// TwinCAT 3 PLC project PLC_SerialCom_Sample1
// ProgramVersion: 3.1.0.8
// libraries:
//   Tc2_SerialCom, * (Beckhoff Automation GmbH)
//   Tc2_Standard, * (Beckhoff Automation GmbH)
//   Tc3_Module, * (Beckhoff Automation GmbH)
// project tree:
//   GVLs/ gc.TcGVL, GVL.TcGVL
//   / PlcTask_Fast.TcTTO (not stored), PlcTask_Standard.TcTTO
//   POUs/ Background.TcPOU, BackgroundKL.TcPOU, BackgroundEL.TcPOU, FB_SerialCom.TcPOU, MAIN.TcPOU, BackgroundPcCOM.TcPOU (not stored), test.TcPOU
// real-time tasks:
//   TASK PlcTask_Fast: cycle T#2ms, priority 19, ADS port 350
//   TASK PlcTask_Standard: cycle T#10ms, priority 20, ADS port 351
// motion (NC):
//   TASK NC-Task 1 SAF: cycle T#2ms, priority 4, ADS port 501
//   TASK NC-Task 1 SVB: cycle T#10ms, priority 8, ADS port 511
//   AXIS Axis 1 (id 1)
//     OtherSettings: AllowMotionCmdToSlave=true
//     encoder EncType=19
//       EncPara: MaxCount=#xffffffff
//     drive DrvType=16
//       DrvPara: MaxCount=#xffffffff, DriveControlDWord=#x00020000
//         Analog: TorqueSetpointScale=10, ScaleFactorActTorque=0.1
//         TimeComp: TaskDelayCycles=1
//     controller CtrType=1
//       CtrPara: PriorControlFactor=1
//         Observer: BandWidth=20
//   AXIS Axis 2 (id 2)
//     OtherSettings: AllowMotionCmdToSlave=true
//     encoder EncType=19
//       EncPara: MaxCount=#xffffffff
//     drive DrvType=16
//       DrvPara: MaxCount=#xffffffff, DriveControlDWord=#x00020000
//         Analog: TorqueSetpointScale=10, ScaleFactorActTorque=0.1
//         TimeComp: TaskDelayCycles=1
//     controller CtrType=1
//       CtrPara: PriorControlFactor=1
//         Observer: BandWidth=20
// I/O:
//   DEVICE Device 1 (COM Port) (disabled)
//   DEVICE Device 3 (EtherCAT) (disabled), AmsNetId 172.17.60.154.4.1
//     Term 1 (EK1100) [EK1100 EtherCAT Coupler (2A E-Bus)]
//       Term 2 (EL6001) [EL6001 Interface (RS232)]
//       Box 3 (BK1250)
//   DEVICE Device 2 (EtherCAT), AmsNetId 192.168.2.2.3.1
//     Term 4 (EK1914) [EK1914, 2 Ch. Safety Input/Output 24V,  TwinSAFE]
//       modules: Module 1 (FSOE), Module 2 (DIO)
//       Term 5 (EL9410) [EL9410 E-Bus Power Supplier  (Diagnostics)]
//       Term 6 (EL3164) [EL3164 4Ch. Ana. Input 0-10V]
//       Term 7 (EL4104) [EL4104 4Ch. Ana. Output 0-10V, 16bit]
//       Term 5 (EL6614) [EL6614 4 Port Switch (Ethernet, CoE)]
//       Term 9 (EL6002) [EL6002 Interface 2Ch. (RS232)]
//       Term 10 (EL9410) [EL9410 E-Bus Power Supplier  (Diagnostics)]
//       Term 11 (EL7201-9014) [EL7201-9014 1Ch. MDP742 Servo motor output stage with OCT (50V, 2.8A RMS) and STO input]
//       Term 12 (EL7201-9014) [EL7201-9014 1Ch. MDP742 Servo motor output stage with OCT (50V, 2.8A RMS) and STO input]
//       Term 10 (EL9011) [EL9011 End Terminal]
// variable links:
//   NC-Task 1 SAF/Axes/Axis 1 <-> Device 2 (EtherCAT)/Term 4 (EK1914)/Term 11 (EL7201-9014)
//     Drive/Inputs/In/nDcOutputTime <-> InfoData/DcOutputShift
//     Drive/Inputs/In/nState1 <-> DRV Statusword/Statusword
//     Drive/Inputs/In/nState2 <-> DRV Statusword/Statusword @bit 8
//     Drive/Inputs/In/nState4 @bit 1 <-> WcState/InputToggle
//     Drive/Inputs/In/nState4 <-> WcState/WcState
//     Drive/Outputs/Out/nCtrl1 <-> DRV Controlword/Controlword
//     Drive/Outputs/Out/nCtrl2 <-> DRV Controlword/Controlword @bit 8
//     Drive/Outputs/Out/nDataOut2 <-> DRV Target velocity/Target velocity
//     Enc/Inputs/In/nDataIn1 <-> FB Position/Position
//     Enc/Inputs/In/nDcInputTime <-> InfoData/DcInputShift
//     Enc/Inputs/In/nState4 @bit 1 <-> WcState/InputToggle
//     Enc/Inputs/In/nState4 <-> WcState/WcState
//   NC-Task 1 SAF/Axes/Axis 2 <-> Device 2 (EtherCAT)/Term 4 (EK1914)/Term 12 (EL7201-9014)
//     Drive/Inputs/In/nDcOutputTime <-> InfoData/DcOutputShift
//     Drive/Inputs/In/nState1 <-> DRV Statusword/Statusword
//     Drive/Inputs/In/nState2 <-> DRV Statusword/Statusword @bit 8
//     Drive/Inputs/In/nState4 @bit 1 <-> WcState/InputToggle
//     Drive/Inputs/In/nState4 <-> WcState/WcState
//     Drive/Outputs/Out/nCtrl1 <-> DRV Controlword/Controlword
//     Drive/Outputs/Out/nCtrl2 <-> DRV Controlword/Controlword @bit 8
//     Drive/Outputs/Out/nDataOut2 <-> DRV Target velocity/Target velocity
//     Enc/Inputs/In/nDataIn1 <-> FB Position/Position
//     Enc/Inputs/In/nDcInputTime <-> InfoData/DcInputShift
//     Enc/Inputs/In/nState4 @bit 1 <-> WcState/InputToggle
//     Enc/Inputs/In/nState4 <-> WcState/WcState
//   PLC_SerialCom_Sample1/PLC_SerialCom_Sample1 Instance <-> Device 2 (EtherCAT)/Term 4 (EK1914)
//     PlcTask_Standard Inputs/test.xTestInput <-> Module 2 (DIO)/DIO Inputs/Input 1
//   PLC_SerialCom_Sample1/PLC_SerialCom_Sample1 Instance <-> Device 2 (EtherCAT)/Term 4 (EK1914)/Term 9 (EL6002)
//     PlcTask_Fast Inputs/BackgroundEL.astIn_EL6002[0]/D <-> COM TxPDO-Map Inputs Channel 1/Data In 0
//     PlcTask_Fast Inputs/BackgroundEL.astIn_EL6002[1]/D <-> COM TxPDO-Map Inputs Channel 2/Data In 0
//     PlcTask_Fast Inputs/BackgroundEL.astIn_EL6002[0]/D @bit 8 <-> COM TxPDO-Map Inputs Channel 1/Data In 1
//     PlcTask_Fast Inputs/BackgroundEL.astIn_EL6002[0]/D @bit 80 <-> COM TxPDO-Map Inputs Channel 1/Data In 10
//     PlcTask_Fast Inputs/BackgroundEL.astIn_EL6002[0]/D @bit 88 <-> COM TxPDO-Map Inputs Channel 1/Data In 11
//     PlcTask_Fast Inputs/BackgroundEL.astIn_EL6002[0]/D @bit 96 <-> COM TxPDO-Map Inputs Channel 1/Data In 12
//     PlcTask_Fast Inputs/BackgroundEL.astIn_EL6002[0]/D @bit 104 <-> COM TxPDO-Map Inputs Channel 1/Data In 13
//     PlcTask_Fast Inputs/BackgroundEL.astIn_EL6002[0]/D @bit 112 <-> COM TxPDO-Map Inputs Channel 1/Data In 14
//     PlcTask_Fast Inputs/BackgroundEL.astIn_EL6002[0]/D @bit 120 <-> COM TxPDO-Map Inputs Channel 1/Data In 15
//     PlcTask_Fast Inputs/BackgroundEL.astIn_EL6002[0]/D @bit 128 <-> COM TxPDO-Map Inputs Channel 1/Data In 16
//     PlcTask_Fast Inputs/BackgroundEL.astIn_EL6002[0]/D @bit 136 <-> COM TxPDO-Map Inputs Channel 1/Data In 17
//     PlcTask_Fast Inputs/BackgroundEL.astIn_EL6002[0]/D @bit 144 <-> COM TxPDO-Map Inputs Channel 1/Data In 18
//     PlcTask_Fast Inputs/BackgroundEL.astIn_EL6002[0]/D @bit 152 <-> COM TxPDO-Map Inputs Channel 1/Data In 19
//     PlcTask_Fast Inputs/BackgroundEL.astIn_EL6002[0]/D @bit 16 <-> COM TxPDO-Map Inputs Channel 1/Data In 2
//     PlcTask_Fast Inputs/BackgroundEL.astIn_EL6002[0]/D @bit 160 <-> COM TxPDO-Map Inputs Channel 1/Data In 20
//     PlcTask_Fast Inputs/BackgroundEL.astIn_EL6002[0]/D @bit 168 <-> COM TxPDO-Map Inputs Channel 1/Data In 21
//     PlcTask_Fast Inputs/BackgroundEL.astIn_EL6002[0]/D @bit 24 <-> COM TxPDO-Map Inputs Channel 1/Data In 3
//     PlcTask_Fast Inputs/BackgroundEL.astIn_EL6002[0]/D @bit 32 <-> COM TxPDO-Map Inputs Channel 1/Data In 4
//     PlcTask_Fast Inputs/BackgroundEL.astIn_EL6002[0]/D @bit 40 <-> COM TxPDO-Map Inputs Channel 1/Data In 5
//     PlcTask_Fast Inputs/BackgroundEL.astIn_EL6002[0]/D @bit 48 <-> COM TxPDO-Map Inputs Channel 1/Data In 6
//     PlcTask_Fast Inputs/BackgroundEL.astIn_EL6002[0]/D @bit 56 <-> COM TxPDO-Map Inputs Channel 1/Data In 7
//     PlcTask_Fast Inputs/BackgroundEL.astIn_EL6002[0]/D @bit 64 <-> COM TxPDO-Map Inputs Channel 1/Data In 8
//     PlcTask_Fast Inputs/BackgroundEL.astIn_EL6002[0]/D @bit 72 <-> COM TxPDO-Map Inputs Channel 1/Data In 9
//     PlcTask_Fast Inputs/BackgroundEL.astIn_EL6002[1]/D @bit 8 <-> COM TxPDO-Map Inputs Channel 2/Data In 1
//     PlcTask_Fast Inputs/BackgroundEL.astIn_EL6002[1]/D @bit 80 <-> COM TxPDO-Map Inputs Channel 2/Data In 10
//     PlcTask_Fast Inputs/BackgroundEL.astIn_EL6002[1]/D @bit 88 <-> COM TxPDO-Map Inputs Channel 2/Data In 11
//     PlcTask_Fast Inputs/BackgroundEL.astIn_EL6002[1]/D @bit 96 <-> COM TxPDO-Map Inputs Channel 2/Data In 12
//     PlcTask_Fast Inputs/BackgroundEL.astIn_EL6002[1]/D @bit 104 <-> COM TxPDO-Map Inputs Channel 2/Data In 13
//     PlcTask_Fast Inputs/BackgroundEL.astIn_EL6002[1]/D @bit 112 <-> COM TxPDO-Map Inputs Channel 2/Data In 14
//     PlcTask_Fast Inputs/BackgroundEL.astIn_EL6002[1]/D @bit 120 <-> COM TxPDO-Map Inputs Channel 2/Data In 15
//     PlcTask_Fast Inputs/BackgroundEL.astIn_EL6002[1]/D @bit 128 <-> COM TxPDO-Map Inputs Channel 2/Data In 16
//     PlcTask_Fast Inputs/BackgroundEL.astIn_EL6002[1]/D @bit 136 <-> COM TxPDO-Map Inputs Channel 2/Data In 17
//     PlcTask_Fast Inputs/BackgroundEL.astIn_EL6002[1]/D @bit 144 <-> COM TxPDO-Map Inputs Channel 2/Data In 18
//     PlcTask_Fast Inputs/BackgroundEL.astIn_EL6002[1]/D @bit 152 <-> COM TxPDO-Map Inputs Channel 2/Data In 19
//     PlcTask_Fast Inputs/BackgroundEL.astIn_EL6002[1]/D @bit 16 <-> COM TxPDO-Map Inputs Channel 2/Data In 2
//     PlcTask_Fast Inputs/BackgroundEL.astIn_EL6002[1]/D @bit 160 <-> COM TxPDO-Map Inputs Channel 2/Data In 20
//     PlcTask_Fast Inputs/BackgroundEL.astIn_EL6002[1]/D @bit 168 <-> COM TxPDO-Map Inputs Channel 2/Data In 21
//     PlcTask_Fast Inputs/BackgroundEL.astIn_EL6002[1]/D @bit 24 <-> COM TxPDO-Map Inputs Channel 2/Data In 3
//     PlcTask_Fast Inputs/BackgroundEL.astIn_EL6002[1]/D @bit 32 <-> COM TxPDO-Map Inputs Channel 2/Data In 4
//     PlcTask_Fast Inputs/BackgroundEL.astIn_EL6002[1]/D @bit 40 <-> COM TxPDO-Map Inputs Channel 2/Data In 5
//     PlcTask_Fast Inputs/BackgroundEL.astIn_EL6002[1]/D @bit 48 <-> COM TxPDO-Map Inputs Channel 2/Data In 6
//     PlcTask_Fast Inputs/BackgroundEL.astIn_EL6002[1]/D @bit 56 <-> COM TxPDO-Map Inputs Channel 2/Data In 7
//     PlcTask_Fast Inputs/BackgroundEL.astIn_EL6002[1]/D @bit 64 <-> COM TxPDO-Map Inputs Channel 2/Data In 8
//     PlcTask_Fast Inputs/BackgroundEL.astIn_EL6002[1]/D @bit 72 <-> COM TxPDO-Map Inputs Channel 2/Data In 9
//     PlcTask_Fast Inputs/BackgroundEL.astIn_EL6002[0]/Status <-> COM TxPDO-Map Inputs Channel 1/Status
//     PlcTask_Fast Inputs/BackgroundEL.astIn_EL6002[1]/Status <-> COM TxPDO-Map Inputs Channel 2/Status
//     PlcTask_Fast Outputs/BackgroundEL.astOut_EL6002[0]/Ctrl <-> COM RxPDO-Map Outputs Channel 1/Ctrl
//     PlcTask_Fast Outputs/BackgroundEL.astOut_EL6002[1]/Ctrl <-> COM RxPDO-Map Outputs Channel 2/Ctrl
//     PlcTask_Fast Outputs/BackgroundEL.astOut_EL6002[0]/D <-> COM RxPDO-Map Outputs Channel 1/Data Out 0
//     PlcTask_Fast Outputs/BackgroundEL.astOut_EL6002[1]/D <-> COM RxPDO-Map Outputs Channel 2/Data Out 0
//     PlcTask_Fast Outputs/BackgroundEL.astOut_EL6002[0]/D @bit 8 <-> COM RxPDO-Map Outputs Channel 1/Data Out 1
//     PlcTask_Fast Outputs/BackgroundEL.astOut_EL6002[0]/D @bit 80 <-> COM RxPDO-Map Outputs Channel 1/Data Out 10
//     PlcTask_Fast Outputs/BackgroundEL.astOut_EL6002[0]/D @bit 88 <-> COM RxPDO-Map Outputs Channel 1/Data Out 11
//     PlcTask_Fast Outputs/BackgroundEL.astOut_EL6002[0]/D @bit 96 <-> COM RxPDO-Map Outputs Channel 1/Data Out 12
//     PlcTask_Fast Outputs/BackgroundEL.astOut_EL6002[0]/D @bit 104 <-> COM RxPDO-Map Outputs Channel 1/Data Out 13
//     PlcTask_Fast Outputs/BackgroundEL.astOut_EL6002[0]/D @bit 112 <-> COM RxPDO-Map Outputs Channel 1/Data Out 14
//     PlcTask_Fast Outputs/BackgroundEL.astOut_EL6002[0]/D @bit 120 <-> COM RxPDO-Map Outputs Channel 1/Data Out 15
//     PlcTask_Fast Outputs/BackgroundEL.astOut_EL6002[0]/D @bit 128 <-> COM RxPDO-Map Outputs Channel 1/Data Out 16
//     PlcTask_Fast Outputs/BackgroundEL.astOut_EL6002[0]/D @bit 136 <-> COM RxPDO-Map Outputs Channel 1/Data Out 17
//     PlcTask_Fast Outputs/BackgroundEL.astOut_EL6002[0]/D @bit 144 <-> COM RxPDO-Map Outputs Channel 1/Data Out 18
//     PlcTask_Fast Outputs/BackgroundEL.astOut_EL6002[0]/D @bit 152 <-> COM RxPDO-Map Outputs Channel 1/Data Out 19
//     PlcTask_Fast Outputs/BackgroundEL.astOut_EL6002[0]/D @bit 16 <-> COM RxPDO-Map Outputs Channel 1/Data Out 2
//     PlcTask_Fast Outputs/BackgroundEL.astOut_EL6002[0]/D @bit 160 <-> COM RxPDO-Map Outputs Channel 1/Data Out 20
//     PlcTask_Fast Outputs/BackgroundEL.astOut_EL6002[0]/D @bit 168 <-> COM RxPDO-Map Outputs Channel 1/Data Out 21
//     PlcTask_Fast Outputs/BackgroundEL.astOut_EL6002[0]/D @bit 24 <-> COM RxPDO-Map Outputs Channel 1/Data Out 3
//     PlcTask_Fast Outputs/BackgroundEL.astOut_EL6002[0]/D @bit 32 <-> COM RxPDO-Map Outputs Channel 1/Data Out 4
//     PlcTask_Fast Outputs/BackgroundEL.astOut_EL6002[0]/D @bit 40 <-> COM RxPDO-Map Outputs Channel 1/Data Out 5
//     PlcTask_Fast Outputs/BackgroundEL.astOut_EL6002[0]/D @bit 48 <-> COM RxPDO-Map Outputs Channel 1/Data Out 6
//     PlcTask_Fast Outputs/BackgroundEL.astOut_EL6002[0]/D @bit 56 <-> COM RxPDO-Map Outputs Channel 1/Data Out 7
//     PlcTask_Fast Outputs/BackgroundEL.astOut_EL6002[0]/D @bit 64 <-> COM RxPDO-Map Outputs Channel 1/Data Out 8
//     PlcTask_Fast Outputs/BackgroundEL.astOut_EL6002[0]/D @bit 72 <-> COM RxPDO-Map Outputs Channel 1/Data Out 9
//     PlcTask_Fast Outputs/BackgroundEL.astOut_EL6002[1]/D @bit 8 <-> COM RxPDO-Map Outputs Channel 2/Data Out 1
//     PlcTask_Fast Outputs/BackgroundEL.astOut_EL6002[1]/D @bit 80 <-> COM RxPDO-Map Outputs Channel 2/Data Out 10
//     PlcTask_Fast Outputs/BackgroundEL.astOut_EL6002[1]/D @bit 88 <-> COM RxPDO-Map Outputs Channel 2/Data Out 11
//     PlcTask_Fast Outputs/BackgroundEL.astOut_EL6002[1]/D @bit 96 <-> COM RxPDO-Map Outputs Channel 2/Data Out 12
//     PlcTask_Fast Outputs/BackgroundEL.astOut_EL6002[1]/D @bit 104 <-> COM RxPDO-Map Outputs Channel 2/Data Out 13
//     PlcTask_Fast Outputs/BackgroundEL.astOut_EL6002[1]/D @bit 112 <-> COM RxPDO-Map Outputs Channel 2/Data Out 14
//     PlcTask_Fast Outputs/BackgroundEL.astOut_EL6002[1]/D @bit 120 <-> COM RxPDO-Map Outputs Channel 2/Data Out 15
//     PlcTask_Fast Outputs/BackgroundEL.astOut_EL6002[1]/D @bit 128 <-> COM RxPDO-Map Outputs Channel 2/Data Out 16
//     PlcTask_Fast Outputs/BackgroundEL.astOut_EL6002[1]/D @bit 136 <-> COM RxPDO-Map Outputs Channel 2/Data Out 17
//     PlcTask_Fast Outputs/BackgroundEL.astOut_EL6002[1]/D @bit 144 <-> COM RxPDO-Map Outputs Channel 2/Data Out 18
//     PlcTask_Fast Outputs/BackgroundEL.astOut_EL6002[1]/D @bit 152 <-> COM RxPDO-Map Outputs Channel 2/Data Out 19
//     PlcTask_Fast Outputs/BackgroundEL.astOut_EL6002[1]/D @bit 16 <-> COM RxPDO-Map Outputs Channel 2/Data Out 2
//     PlcTask_Fast Outputs/BackgroundEL.astOut_EL6002[1]/D @bit 160 <-> COM RxPDO-Map Outputs Channel 2/Data Out 20
//     PlcTask_Fast Outputs/BackgroundEL.astOut_EL6002[1]/D @bit 168 <-> COM RxPDO-Map Outputs Channel 2/Data Out 21
//     PlcTask_Fast Outputs/BackgroundEL.astOut_EL6002[1]/D @bit 24 <-> COM RxPDO-Map Outputs Channel 2/Data Out 3
//     PlcTask_Fast Outputs/BackgroundEL.astOut_EL6002[1]/D @bit 32 <-> COM RxPDO-Map Outputs Channel 2/Data Out 4
//     PlcTask_Fast Outputs/BackgroundEL.astOut_EL6002[1]/D @bit 40 <-> COM RxPDO-Map Outputs Channel 2/Data Out 5
//     PlcTask_Fast Outputs/BackgroundEL.astOut_EL6002[1]/D @bit 48 <-> COM RxPDO-Map Outputs Channel 2/Data Out 6
//     PlcTask_Fast Outputs/BackgroundEL.astOut_EL6002[1]/D @bit 56 <-> COM RxPDO-Map Outputs Channel 2/Data Out 7
//     PlcTask_Fast Outputs/BackgroundEL.astOut_EL6002[1]/D @bit 64 <-> COM RxPDO-Map Outputs Channel 2/Data Out 8
//     PlcTask_Fast Outputs/BackgroundEL.astOut_EL6002[1]/D @bit 72 <-> COM RxPDO-Map Outputs Channel 2/Data Out 9

CONFIGURATION PLC_SerialCom_Sample1
    RESOURCE PLC ON TwinCAT3
        TASK PlcTask_Standard(INTERVAL := T#10ms, PRIORITY := 20);
        PROGRAM MAIN WITH PlcTask_Standard : MAIN;
        PROGRAM test WITH PlcTask_Standard : test;
    END_RESOURCE
END_CONFIGURATION

// ---- GVLs/gc.TcGVL
{attribute 'qualified_only'}
VAR_GLOBAL CONSTANT
	MINDEVICEINDEX				: USINT	:= 0; //on EL6002
	MAXDEVICEINDEX				: USINT	:= 1; //on EL6002
	EL6002_INDEX1				: USINT	:= 0;
	EL6002_INDEX2				: USINT	:= 1;
END_VAR

// ---- GVLs/GVL.TcGVL
VAR_GLOBAL
	aRxBufferEL			: ARRAY[gc.MINDEVICEINDEX..gc.MAXDEVICEINDEX] OF ComBuffer;	(* Receive data buffer; used with all receive function blocks *)
	aTxBufferEL			: ARRAY[gc.MINDEVICEINDEX..gc.MAXDEVICEINDEX] OF ComBuffer;	(* Transmit data buffer; used with all receive function blocks *)

//	RxBufferKL			: ComBuffer;	(* Receive data buffer; used with all receive function blocks *)
//	TxBufferKL			: ComBuffer;	(* Transmit data buffer; used with all receive function blocks *)
END_VAR

// ---- POUs/MAIN.TcPOU
(*
SerialCom_InfoSys_Sample1 (v2.0)
This sample sends and receives a string via serial communication.
Three hardware interfaces are used: Pc COM port, EL terminal, KL terminal
*)
PROGRAM MAIN
VAR
//	fbPcCom		: FB_SerialCom;
	afbEL6002	: ARRAY[gc.MINDEVICEINDEX..gc.MAXDEVICEINDEX] OF FB_SerialCom;
//	fbKL6001	: FB_SerialCom;
	
	(* exchange buffers with background communication with the PC COM port device *)
//	RxBufferPcCom	: ComBuffer;	(* Receive data buffer; used with all receive function blocks *)
//	TxBufferPcCom	: ComBuffer;	(* Transmit data buffer; used with all receive function blocks *)
END_VAR

(* background communication with the PC COM port device *)
//BackgroundPcCOM(RxBufferPcCom:=RxBufferPcCom, TxBufferPcCom:=TxBufferPcCom);

(* Send and receive commands *)
//fbPcCom(TxBuffer:=TxBufferPcCom, RxBuffer:=RxBufferPcCom);

//fbKL6001(TxBuffer:=TxBufferKL, RxBuffer:=RxBufferKL);

afbEL6002[gc.EL6002_INDEX1](TxBuffer:=aTxBufferEL[gc.EL6002_INDEX1], RxBuffer:=aRxBufferEL[gc.EL6002_INDEX1]);

afbEL6002[gc.EL6002_INDEX2](TxBuffer:=aTxBufferEL[gc.EL6002_INDEX2], RxBuffer:=aRxBufferEL[gc.EL6002_INDEX2]);

END_PROGRAM

// ---- POUs/FB_SerialCom.TcPOU
FUNCTION_BLOCK FB_SerialCom
VAR_IN_OUT
	TxBuffer	: ComBuffer;
	RxBuffer	: ComBuffer;
END_VAR
VAR
	Timer		: TON := (PT:=T#1S);
	fbSend		: SendString;
	bSendBusy	: BOOL;
	eSendErrorID: ComError_t;

	fbReceive		: ReceiveString;
	sReceivedString	: STRING;
	sLastReceivedString: STRING;
	bStringReceived	: BOOL;
	bReceiveBusy	: BOOL;
	bReceiveError	: BOOL;
	eReceiveErrorID	: ComError_t;
	bReceiveTimeout	: BOOL;
	nReceiveCounter	: UDINT;
END_VAR
VAR_OUTPUT
		
END_VAR

// Call the send block every second to repeat the transmission.
// Also call the block as long as it is busy to finish a transmission.
Timer(IN:=TRUE);
IF Timer.Q OR fbSend.Busy THEN
	Timer(IN:=FALSE); (* reset timer *)
	fbSend(	SendString:= '$02Hello World ! $03',
			TXbuffer:= TxBuffer,
			Busy=> bSendBusy,
			Error=> );
	IF fbSend.Error <> COMERROR_NOERROR THEN
		eSendErrorID := fbSend.Error;
	END_IF
END_IF

//	Receive string data:
//	The block receives any data strings beginning with a STX ($02) and ending with an ETX ($03) character.	
fbReceive(
	Prefix:= '$02',
	Suffix:= '$03',
	Timeout:= T#1s,
	ReceivedString:= sReceivedString,
	Rxbuffer:= RxBuffer,
	StringReceived=> bStringReceived,
	Busy=> bReceiveBusy,
	Error=> ,
	RxTimeout=> bReceiveTimeout );
IF fbReceive.Error <> COMERROR_NOERROR THEN
	eReceiveErrorID := fbReceive.Error;
END_IF
IF bStringReceived THEN
	nReceiveCounter := nReceiveCounter + 1;
	sLastReceivedString := sReceivedString;
END_IF

END_FUNCTION_BLOCK

// ---- POUs/test.TcPOU
PROGRAM test
VAR
	xTestInput	AT %I* : BOOL;
END_VAR

END_PROGRAM

// ---- POUs/Background.TcPOU
PROGRAM Background
VAR
END_VAR

(*
The SerialLineControl function block is supposed to be called in every PLC cycle.
It communicates with the serial line hardware device and transmits or receives data.
The SerialLineControl can be called in the standard task (e.g.for PcCOM port usage) 
or in a separate fast task (e.g.for terminal usage) as well.
A fast separate task will be necessary at high baud rates or with KL6001 terminals 
which have a small process image (3 or 5 data bytes only)
*)

(* background communication with the EL6001 terminal *)
BackgroundEL();

(* background communication with the KL6001 terminal (3byte) *)
//BackgroundKL();

END_PROGRAM

// ---- POUs/BackgroundEL.TcPOU
PROGRAM BackgroundEL
VAR
	(* background communication with the EL6001/EL6002 terminal *)
	afbEL6002Ctrl			: ARRAY[gc.MINDEVICEINDEX..gc.MAXDEVICEINDEX] OF SerialLineControl;
	abEL6002CtrlError		: ARRAY[gc.MINDEVICEINDEX..gc.MAXDEVICEINDEX] OF BOOL;
	aeEL6002CtrlErrorID		: ARRAY[gc.MINDEVICEINDEX..gc.MAXDEVICEINDEX] OF ComError_t;
	(* 	I/O variables for a EL6001 terminal*)
	astIn_EL6002 AT %I*		: ARRAY[gc.MINDEVICEINDEX..gc.MAXDEVICEINDEX] OF EL6inData22B;	(* linked to the EL6001 in the TwinCAT System Manager *)
	astOut_EL6002 AT %Q*	: ARRAY[gc.MINDEVICEINDEX..gc.MAXDEVICEINDEX] OF EL6outData22B;(* linked to the EL6001 in the TwinCAT System Manager *)
END_VAR

(*
The SerialLineControl function block is supposed to be called in every PLC cycle.
It communicates with the serial line hardware device and transmits or receives data.
The SerialLineControl can be called in the standard task (e.g.for PcCOM port usage) 
or in a separate fast task (e.g.for terminal usage) as well.
A fast separate task will be necessary at high baud rates or with KL6001 terminals 
which have a small process image (3 or 5 data bytes only)
*)

(* background communication with the EL6002 terminal *)

//use with type SerialLineControl
afbEL6002Ctrl[gc.EL6002_INDEX1](
	Mode:= SERIALLINEMODE_EL6_22B, 
	pComIn:= ADR(astIn_EL6002[gc.EL6002_INDEX1]), 
	pComOut:= ADR(astOut_EL6002[gc.EL6002_INDEX1]), 
	SizeComIn:= SIZEOF(astIn_EL6002[gc.EL6002_INDEX1]), 
	Error=> , 
	ErrorID=> , 
	TxBuffer:= aTxBufferEL[gc.EL6002_INDEX1], 
	RxBuffer:= aRxBufferEL[gc.EL6002_INDEX1] );
IF afbEL6002Ctrl[gc.EL6002_INDEX1].Error THEN
	abEL6002CtrlError[gc.EL6002_INDEX1] := TRUE;
	aeEL6002CtrlErrorID[gc.EL6002_INDEX1] := afbEL6002Ctrl[gc.EL6002_INDEX1].ErrorID;
END_IF

END_PROGRAM

// ---- POUs/BackgroundKL.TcPOU
PROGRAM BackgroundKL
VAR
	(* background communication with the KL6001 terminal (3byte) *)
	fbKL6001Ctrl		: SerialLineControl;
	bKL6001CtrlError	: BOOL;
	eKL6001CtrlErrorID	: ComError_t;
	fbKL6001Config		: KL6configuration;
	bKL6001ConfigError	: BOOL;
	eKL6001ConfigErrorID: ComError_t;
	bKL6001ConfigExe	: BOOL := TRUE;
	(* 	I/O variables for a KL6001 terminal*)
	stIn_KL6001 AT %I*	: KL6inData;	(* linked to the KL6001 in the TwinCAT System Manager *)
	stOut_KL6001 AT %Q*	: KL6outData;	(* linked to the KL6001 in the TwinCAT System Manager *)
END_VAR

(*
The SerialLineControl function block is supposed to be called in every PLC cycle.
It communicates with the serial line hardware device and transmits or receives data.
The SerialLineControl can be called in the standard task (e.g.for PcCOM port usage) 
or in a separate fast task (e.g.for terminal usage) as well.
A fast separate task will be necessary at high baud rates or with KL6001 terminals 
which have a small process image (3 or 5 data bytes only)
*)
(*
(* background communication with the KL6001 terminal (3byte) *)
fbKL6001Config(
	Execute:= bKL6001ConfigExe, 
	Mode:= SERIALLINEMODE_KL6_3B_ALTERNATIVE, 
	Baudrate:= 9600, 
	NoDatabits:= 8, 
	Parity:= 0, 
	Stopbits:= 1, 
	Handshake:= HANDSHAKE_NONE, 
	ContinousMode:= FALSE, 
	pComIn:= ADR(stIn_KL6001), 
	pComOut:= ADR(stOut_KL6001), 
	SizeComIn:= SIZEOF(stIn_KL6001), 
	Done=> , 
	Busy=> , 
	Error=> , 
	ErrorId=>  );
IF fbKL6001Config.Error THEN
	bKL6001ConfigError := TRUE;
	eKL6001ConfigErrorID := fbKL6001Config.ErrorId;
END_IF
	
IF NOT fbKL6001Config.Busy AND NOT bKL6001ConfigError THEN
	bKL6001ConfigExe := FALSE;
	fbKL6001Ctrl(
		Mode:= SERIALLINEMODE_KL6_3B_ALTERNATIVE,
		pComIn:= ADR(stIn_KL6001),
		pComOut:= ADR(stOut_KL6001),
		SizeComIn:= SIZEOF(stIn_KL6001),
		Error=> ,
		ErrorID=> ,
		TxBuffer:= TxBufferKL,
		RxBuffer:= RxBufferKL );
	IF fbKL6001Ctrl.Error THEN
		bKL6001CtrlError := TRUE;
		eKL6001CtrlErrorID := fbKL6001Ctrl.ErrorID;
	END_IF
END_IF
*)

END_PROGRAM
